FUNCTION AddNums : INT
VAR_INPUT
	fbMotor1 : Motor;
END_VAR
VAR
END_VAR


IF __ISVALIDREF(fbMotor1) THEN
	AddNums := 1;
END_IF

END_FUNCTION

(* stored: Version 1.1.0.1, ProductVersion 3.1.4024.16
   POU AddNums: Id {63e600e2-a8d3-4326-9584-5f1f91a7a69d}, SpecialFunc None *)
